FUNCTION_BLOCK Await IMPLEMENTS Awaitable

VAR_OUTPUT
END_VAR
VAR
	step: POINTER TO UDINT;
	oldStep: UDINT;
	
	errorCatched: BOOL;
	errorRaised: BOOL;
	increaseByValue: UDINT;

	errorCounter: UDINT;
	errorNames : ARRAY [0..cMax] OF STRING;
	errorMessages : ARRAY [0..cMax] OF STRING;
END_VAR
VAR CONSTANT
    cMax    : UDINT := 1000;
END_VAR

METHOD call : Awaitable
VAR_INPUT
	callback: Callback;
END_VAR
call := THIS^;

IF NOT errorRaised
	AND callback <> 0
	THEN
	
	callback.execute();
	
END_IF
END_METHOD

METHOD catchIf : Awaitable
VAR_INPUT
	error: BOOL;
	callback: REFERENCE TO AwaitableError;
	message: STRING(255);
END_VAR
catchIf := THIS^;

IF errorRaised
	THEN
	RETURN;
END_IF

THIS^.errorCatched := THIS^.errorCatched OR error;

IF error
	THEN
	onError(callback, message, 0);
END_IF
END_METHOD

METHOD continueIf : Awaitable
VAR_INPUT
	value: BOOL;
END_VAR
continueIf := THIS^;

// Make sure step is a valid pointer
IF step = 0 
	OR errorRaised
	THEN
	RETURN;
END_IF


IF value AND NOT THIS^.errorCatched
	THEN
	
	step^ := step^ + increaseByValue;

END_IF
END_METHOD

METHOD evalue : Awaitable
VAR_INPUT
	value: BOOL;
	onTrueCallback: Callback;
	onFalseCallback: REFERENCE TO AwaitableError;
	message: STRING(255);
END_VAR
evalue := THIS^;

// Make sure step is a valid pointer
IF step = 0 
	OR errorRaised
	THEN
	RETURN;
END_IF


IF value AND NOT THIS^.errorCatched
	THEN
	
	step^ := step^ + increaseByValue;
	
	IF onTrueCallback <> 0
	THEN
		onTrueCallback.execute();
	END_IF
	
ELSIF NOT value 
	THEN
	onError(onFalseCallback, message, errorCatched);
END_IF
END_METHOD

METHOD PRIVATE onError : PVOID
VAR_INPUT
	callback: REFERENCE TO AwaitableError;
	message: STRING(255);
	errorRef: REFERENCE TO BOOL;
END_VAR
IF __ISVALIDREF(errorRef)
	THEN
	errorRef := TRUE;
END_IF

	
IF __ISVALIDREF(callback)
	THEN
	
	callback.errorMessage := message;
	IF errorCounter <= cMax
		THEN
		errorNames[errorCounter] := callback.getName();
		errorMessages[errorCounter] := callback.getMessage();
		errorCounter := errorCounter + 1;
	END_IF

	oldStep := step^; 
	step^ := callback.execute();
	
END_IF
END_METHOD

METHOD raiseIf : Awaitable
VAR_INPUT
	error: BOOL;
	callback: REFERENCE TO AwaitableError;
	message: STRING(255);
END_VAR
raiseIf := THIS^;

IF errorRaised
	THEN
	RETURN;
END_IF

IF error 
	THEN
	onError(callback, message, errorRaised);
END_IF
END_METHOD

METHOD reset : PVOID
VAR_INPUT
END_VAR

VAR
	i: UDINT;
END_VAR
errorCounter := 0;
FOR i := 0 TO THIS^.cMAX DO
	IF errorNames[i] = ''
		THEN
		EXIT;
	END_IF
    errorNames[i] := '';
	errorMessages[i] := '';
END_FOR 


errorCatched := FALSE;
errorRaised := FALSE;
oldStep := 0;
END_METHOD

PROPERTY setIncreaseValue : UDINT
SET
increaseByValue := setIncreaseValue;
END_SET
END_PROPERTY

PROPERTY PUBLIC setStepPointer : POINTER TO UDINT
SET
step := setStepPointer;
END_SET
END_PROPERTY

END_FUNCTION_BLOCK

(* stored: Version 1.1.0.1, ProductVersion 3.1.4024.12
   POU Await: Id {16e3a70a-96d3-439c-843d-a8d9992b6297}, SpecialFunc None
   Method call: Id {786c2cbe-5d6b-46ec-bdf3-537e82819b3a}
   Method catchIf: Id {25a4749c-003d-485a-bcd3-c44d5041ff62}
   Method continueIf: Id {d30e2228-9054-4343-8666-4a54ca7559ee}
   Method evalue: Id {6241a87e-533a-4623-a880-40111779f1ee}
   Method onError: Id {2c3cdcfe-3a34-4051-874e-ca50a4da7e63}
   Method raiseIf: Id {2e998d0f-01ef-4e26-ac7c-f91b5e39aaaf}
   Method reset: Id {f9c1e191-47fe-4cf4-a6df-939c24fcccf6}
   Property setIncreaseValue: Id {486e4629-2a04-4991-8f81-a43edd17cbe4}
   Set Set: Id {b007a068-445b-4984-83a9-112f4a9d34f2}
   Property setStepPointer: Id {7bba5888-3f5c-4c1a-b0ea-8945ac6896ed}
   Set Set: Id {bc50a8ff-1df7-456f-90d3-3e094d144b56} *)
